// TIA Portal project "práctica 22ç" (V15)

(* hardware
DEVICE "S7-1200 station_1"  S7-1200 Station
   slot 0: "Rack_0"  S7-1200 Rack  Rack  V1.0
   slot 1: "PLC_1"  CPU 1214C AC/DC/Rly  6ES7 214-1BG40-0XB0  V4.2
*)

// ===== PLC "PLC_1"  CPU 1214C AC/DC/Rly =====

VAR_GLOBAL   // PLC tag table "Tabla de variables estándar"
   "System_Byte" AT %MB254 : Byte;
   "FirstScan" AT %M254.0 : Bool;
   "DiagStatusUpdate" AT %M254.1 : Bool;
   "AlwaysTRUE" AT %M254.2 : Bool;
   "AlwaysFALSE" AT %M254.3 : Bool;
   "Clock_Byte" AT %MB255 : Byte;
   "Clock_10Hz" AT %M255.0 : Bool;
   "Clock_5Hz" AT %M255.1 : Bool;
   "Clock_2.5Hz" AT %M255.2 : Bool;
   "Clock_2Hz" AT %M255.3 : Bool;
   "Clock_1.25Hz" AT %M255.4 : Bool;
   "Clock_1Hz" AT %M255.5 : Bool;
   "Clock_0.625Hz" AT %M255.6 : Bool;
   "Clock_0.5Hz" AT %M255.7 : Bool;
   "Marca" AT %M30.0 : Bool;   // Marca de la interrupción
   "desactiva la marca" AT %I0.6 : Bool;
   "Tag_1" AT %I0.4 : Bool;
   "Tag_2" AT %I0.5 : Bool;
   "LED 1" AT %Q0.6 : Bool;
   "LED 2" AT %Q0.7 : Bool;
END_VAR

ORGANIZATION_BLOCK "Main"   // OB1, LAD, ProgramCycle
TITLE = "Main Program Sweep (Cycle)"
{ S7_Optimized_Access := 'TRUE' }
VERSION : 0.1
   VAR_INPUT
      Initial_Call : Bool;   // Initial call of this OB
      Remanence : Bool;   // =True, if remanent data are available
   END_VAR
BEGIN

REGION Network 1
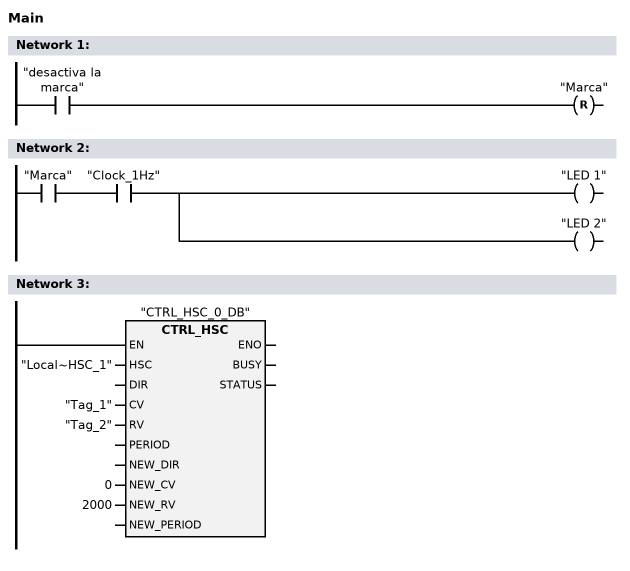
   RUNG wire#powerrail
      Contact( "desactiva la marca" )
      R_Coil( "Marca" )
   END_RUNG
   // the same network as SCL:
   IF "desactiva la marca" THEN "Marca" := FALSE; END_IF;
END_REGION

REGION Network 2
   RUNG wire#powerrail
      Contact( "Marca" )
      Contact( "Clock_1Hz" )
      wire#w1
      Coil( "LED 1" )
   END_RUNG
   RUNG wire#w1
      Coil( "LED 2" )
   END_RUNG
   // the same network as SCL:
   "LED 1" := "Marca" AND "Clock_1Hz";
   "LED 2" := "LED 1";
END_REGION

REGION Network 3
   "CTRL_HSC_0_DB"(HSC := "Local~HSC_1", CV := "Tag_1", RV := "Tag_2", NEW_CV := 0, NEW_RV := 2000);   // CTRL_HSC
END_REGION
END_ORGANIZATION_BLOCK

ORGANIZATION_BLOCK "Hardware interrupt"   // OB40, LAD, HWProcessInterrupt
{ S7_Optimized_Access := 'TRUE' }
VERSION : 0.1
   VAR_INPUT
      LADDR : Hw_Io;   // Hardware identifier
      USI : Word;   // User structure identifier
      IChannel : USInt;   // Interrupt channel number
      EventType : Byte;   // EventType
   END_VAR
BEGIN

REGION Network 1: Marca de la interrupción
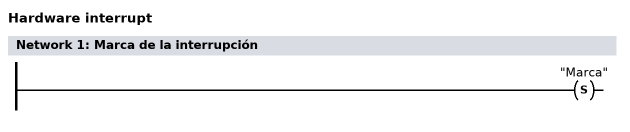
   RUNG wire#powerrail
      S_Coil( "Marca" )
   END_RUNG
   // the same network as SCL:
   "Marca" := TRUE;
END_REGION
END_ORGANIZATION_BLOCK